(* Logix 5000 project; controller BreakGroup_US vendor 1 type 14 code 211 rev 32.16; software revision 32.05; part 2 of 8 *)

VAR_GLOBAL   (* controller tags *)
   Emg_Stop : BOOL;
   Gantry_01Vertical_Limit_Switch_1 : ALIAS FOR MCP_PT01:23:I.0;
   Gantry_01Vertical_Limit_Switch_2 : ALIAS FOR MCP_PT01:23:I.1;
   Gantry_02_Vertical_Limit_Switch_1 : ALIAS FOR RCP_PT01:22:I.7;
   Gantry_02_Vertical_Limit_Switch_2 : ALIAS FOR RCP_PT01:23:I.0;
   Gantry_1_Clamping_Start_PB : ALIAS FOR MCP_PT01:24:I.5;
   Gantry_1_Clamping_Stop_PB : ALIAS FOR MCP_PT01:24:I.6;
   Gantry_1_EMG_PB : ALIAS FOR MCP_PT01:24:I.0;
   Gantry_1_Gripper_Start : BOOL;
   Gantry_1_Home_PB : ALIAS FOR MCP_PT01:24:I.7;
   Gantry_1_Horizontal_Limit_Switch_01 : ALIAS FOR MCP_PT01:22:I.4;
   Gantry_1_Horizontal_Limit_Switch_02 : ALIAS FOR MCP_PT01:22:I.5;
   Gantry_1_Horizontal_Start : BOOL;
   Gantry_1_Horizontal_Start_PB : ALIAS FOR MCP_PT01:24:I.1;
   Gantry_1_Horizontal_Stop_PB : ALIAS FOR MCP_PT01:24:I.2;
   Gantry_1_LH_Clamping_Limit_Switch_1 : ALIAS FOR MCP_PT01:23:I.2;
   Gantry_1_LH_Clamping_Limit_Switch_2 : ALIAS FOR MCP_PT01:23:I.3;
   Gantry_1_RH_Clamping_Limit_Switch_1 : ALIAS FOR MCP_PT01:23:I.4;
   Gantry_1_RH_Clamping_Limit_Switch_2 : ALIAS FOR MCP_PT01:23:I.5;
   Gantry_1_Vertical_Locking_Cyl_1Extended : ALIAS FOR MCP_PT01:23:I.6;
   Gantry_1_Vertical_Locking_Cyl_1Retracted : ALIAS FOR MCP_PT01:23:I.7;
   Gantry_1_Vertical_Start : BOOL;
   Gantry_1_Vertical_Start_PB : ALIAS FOR MCP_PT01:24:I.3;
   Gantry_1_Vertical_Stop_PB : ALIAS FOR MCP_PT01:24:I.4;
   Gantry_1Collision_sensor : ALIAS FOR MCP_PT01:22:I.6;
   Gantry_1Zero_Pos_Sensor : ALIAS FOR MCP_PT01:22:I.7;
   Gantry_2_Clamping_Start_PB : ALIAS FOR RCP_PT01:24:I.6;
   Gantry_2_Clamping_Stop_PB : ALIAS FOR RCP_PT01:24:I.7;
   Gantry_2_Collision_sensor : ALIAS FOR RCP_PT01:22:I.5;
   Gantry_2_Emg_PB : ALIAS FOR RCP_PT01:24:I.1;
   Gantry_2_Gripper_Start : BOOL;
   Gantry_2_Horizontal_Limit_Switch_01 : ALIAS FOR RCP_PT01:22:I.3;
   Gantry_2_Horizontal_Limit_Switch_02 : ALIAS FOR RCP_PT01:22:I.4;
   Gantry_2_Horizontal_Start : BOOL;
   Gantry_2_Horizontal_Start_PB : ALIAS FOR RCP_PT01:24:I.2;
   Gantry_2_Horizontal_Stop_PB : ALIAS FOR RCP_PT01:24:I.3;
   Gantry_2_LH_Clamping_Limit_Switch_1 : ALIAS FOR RCP_PT01:23:I.1;
   Gantry_2_LH_Clamping_Limit_Switch_2 : ALIAS FOR RCP_PT01:23:I.2;
   Gantry_2_LH_Tilting_Home_PositionSensor : ALIAS FOR RCP_PT01:23:I.7;
   Gantry_2_RH_Clamping_Limit_Switch_1 : ALIAS FOR RCP_PT01:23:I.3;
   Gantry_2_RH_Clamping_Limit_Switch_2 : ALIAS FOR RCP_PT01:23:I.4;
   Gantry_2_RH_Tilting_Home_PositionSensor : ALIAS FOR RCP_PT01:24:I.0;
   Gantry_2_Tilter_LH_Start : BOOL;
   Gantry_2_Tilter_RH_Start : BOOL;
   Gantry_2_Vertical_Locking_Cyl_1Extended : ALIAS FOR RCP_PT01:23:I.5;
   Gantry_2_Vertical_Locking_Cyl_1Retracted : ALIAS FOR RCP_PT01:23:I.6;
   Gantry_2_vertical_Start : BOOL;
   Gantry_2_Vertical_Start_PB : ALIAS FOR RCP_PT01:24:I.4;
   Gantry_2_Vertical_Stop_PB : ALIAS FOR RCP_PT01:24:I.5;
   Gantry_2_Zero_Pos_Sensor : ALIAS FOR RCP_PT01:22:I.6;
   HMI_ACK : BOOL;
   HMI_Gantry_01_Gripper_PB : SINT;
   HMI_Gantry_01_Hor_PB : SINT;
   HMI_Gantry_01_Ver_PB : SINT;
   HMI_Gantry_02_Hor_PB : SINT;
        .0   // Gantry_02_horizontal axis servo enable
        .1   // gantry 2 horizontal axis jog mode selected
        .2   // gantry 2 horizontal axis abs mode selected
        .3   // gantry 2 horizontal axis rel mode selected
        .4   // gantry 2 horizontal start command
        .5   // gantry 2 horizontal axis jog forward cmnd
        .6   // gantry 2 horizontal axis jog reverse cmnd
   HMI_Gantry_2_gripper_PB : SINT;
        .0   // Gantry_2_gripper axis servo enable
        .1   // Gantry_2_gripper axis jog mode selected
        .2   // Gantry_2_gripper axis pos mode selected
        .3   // Gantry_2_gripper axis rel mode selected
        .4   // Gantry_2_gripper axis start command
        .5   // Gantry_2_gripper axis jog forward command
        .6   // Gantry_2_gripper axis jog reverse command
   HMI_Gantry_2_Tilter_LH_PB : SINT;
        .0   // Gantry_2_Tilter_LH axis servo enable
        .1   // Gantry_2_Tilter_LH axis jog mode selected
        .2   // Gantry_2_Tilter_LH axis pos mode selected
        .3   // Gantry_2_Tilter_LH axis rel mode selected
        .4   // Gantry_2_Tilter_LH axis start command
        .5   // Gantry_2_Tilter_LH axis jog forward command
        .6   // Gantry_2_Tilter_LH axis jog reverse command
   HMI_Gantry_2_Tilter_RH_PB : SINT;
        .0   // Gantry_2_Tilter_RH axis servo enable
        .1   // Gantry_2_Tilter_RH axis jog mode selected
        .2   // Gantry_2_Tilter_RH pos mode selected
        .3   // Gantry_2_Tilter_RH rel mode selected
        .4   // Gantry_2_Tilter_RH axis start command
        .5   // Gantry_2_Tilter_RH axis jog forward command
        .6   // Gantry_2_Tilter_RH axis jog rev command
   HMI_Gantry_2_vertical_PB : SINT;
        .0   // Gantry_2_vertical axis servo enable
        .1   // Gantry_2_vertical axis jog mode selected
        .2   // Gantry_2_vertical axis pos mode selected
        .3   // Gantry_2_vertical axis rel mode selected
        .4   // Gantry_2_vertical start command
        .5   // Gantry_2_vertical axis jog forward command
        .6   // Gantry_2_vertical axis jog reverse command
   HMI_MAN_GTY1_GRI_STOP : BOOL;
   HMI_MAN_GTY1_HORIZ_STOP : BOOL;
   HMI_MAN_GTY1_VERT_STOP : BOOL;
   HMI_MAN_GTY2_GRI_STOP : BOOL;
   HMI_MAN_GTY2_HORI_STOP : BOOL;
   HMI_MAN_GTY2_TIL1_STOP : BOOL;
   HMI_MAN_GTY2_TIL2_STOP : BOOL;
   HMI_MAN_GTY2_VERT_STOP : BOOL;
   HMI_MAN_LH_OIL_STOP : BOOL;
   HMI_MAN_RH_OIL_STOP : BOOL;
   HMI_MAN_STN_100_STOP : BOOL;
   HMI_MAN_STN_110_STOP : BOOL;
   HMI_MAN_STN_120_STOP : BOOL;
   HMI_MAN_STN_30_STOP : BOOL;
   HMI_MAN_STN_40_STOP : BOOL;
   HMI_MAN_STN_50_STOP : BOOL;
   HMI_MAN_STN_60_STOP : BOOL;
   HMI_MAN_STN_70_STOP : BOOL;
   HMI_MAN_STN_80_STOP : BOOL;
   HMI_MAN_STN_90_STOP : BOOL;
   HMI_Oil_Tank_LH_PB : SINT;
   HMI_Oil_Tank_RH_PB : SINT;
   HMI_STN30_GRI_SETPOINT : REAL := 300.0;
   HMI_STN30_HORIZ_MOVE_SETPOINT : REAL := 2000.0;
   HMI_STN30_VER_LIFTUP_SETPOINT : REAL := 10.0;
   HMI_STN30_VER_PICK_SETPOINT : REAL := 50.0;
   HMI_STN40_GRI_GRIP_POINT : REAL;
   HMI_STN40_GRI_SETPOINT : REAL := 200.0;
   HMI_STN40_HORIZ_MOVE_SETPOINT : REAL := 1000.0;
   HMI_STN40_VER_LIFTUP_SETPOINT : REAL := 10.0;
   HMI_STN40_VER_PICK_LIFTUP_SETPOINT : REAL;
   HMI_STN40_VER_PICK_SETPOINT : REAL := 50.0;
   HMI_STN40_VER_PLACE_SETPOINT : REAL;
   HMI_STN50_DE_GRIPPER_SETPOINT : REAL;
   HMI_STN50_GRI_GRIP_POINT : REAL;
   HMI_STN50_HORIZ_MOVE_SETPOINT : REAL;
   HMI_STN50_VER_DROP_SETPOINT : REAL;
   HMI_STN50_VER_LIFTUP_SETPOINT : REAL;
   HMI_STN50_VER_PICK_LIFTUP_SETPOINT : REAL;
   HMI_STN50_VER_PICK_SETPOINT : DINT;
   MAN_GTY1_GRI_HOME : TIMER := (PRE := 1000);
   MAN_GTY1_HORI_HOME : TIMER := (PRE := 1000);
   MAN_GTY1_VERT_HOME : TIMER := (PRE := 1000);
   MAN_GTY2_GRI_HOME : TIMER := (PRE := 1000);
   MAN_GTY2_HORI_HOME : TIMER := (PRE := 1000);
   MAN_GTY2_TIL1_HOME : TIMER := (PRE := 1000);
   MAN_GTY2_TIL2_HOME : TIMER := (PRE := 1000);
   MAN_GTY2_VERT_HOME : TIMER := (PRE := 1000);
   MAN_LH_OIL_TIME : TIMER := (PRE := 1000);
   MAN_RH_OIL_TIME : TIMER := (PRE := 1000);
   MAN_STN_100_HOME : TIMER := (PRE := 1000);
   MAN_STN_110_HOME : TIMER := (PRE := 1000);
   MAN_STN_120_HOME : TIMER := (PRE := 1000);
   MAN_STN_30_HOME : TIMER := (PRE := 1000);
   MAN_STN_40_HOME : TIMER := (PRE := 1000);
   MAN_STN_50_HOME : TIMER := (PRE := 1000);
   man_STN_60_HOME : TIMER := (PRE := 1000);
   MAN_STN_70_HOME : TIMER := (PRE := 1000);
   MAN_STN_80_HOME : TIMER := (PRE := 1000);
   MAN_STN_90_HOME : TIMER := (PRE := 1000);
   MCP_GY_01_Gripper : MCP_Servo_01 := (Inverter_Ready := 1, STO_InActive := 1, Referenced_Drive := 1, Status_Suberror_Num := 13, Digital_Inputs := 2#0000_0000_0000_0001, Actual_Mode := 400, Actual_Pos := 331.5, Enable_EsTop := 1, Speed := 10.0, Accel_Ramp := 30.0, Decel_Ramp := 30.0, Application_Mode := 400, Target_Position := 331.5, PositionDecimal_Place := 2);
   MCP_GY_01_Horizontal : MCP_Servo_02 := (Start_Offest_Num := 16, Inverter_Ready := 1, STO_InActive := 1, Referenced_Drive := 1, SftWreLiMits_DisAble := 1, Status_Suberror_Num := 13, Digital_Inputs := 2#0000_0000_0000_0001, Actual_Mode := 400, Actual_Pos := 6159.3, Enable_EsTop := 1, Speed := 20.0, Accel_Ramp := 100.0, Decel_Ramp := 100.0, Application_Mode := 400, Target_Position := 6159.3, PositionDecimal_Place := 2);
   MCP_GY_01_Vertical : MCP_Servo_02 := (Start_Offest_Num := 8, Inverter_Ready := 1, STO_InActive := 1, Referenced_Drive := 1, Status_Suberror_Num := 13, Digital_Inputs := 2#0000_0000_0000_0001, Actual_Mode := 400, Actual_Pos := 570.8, Enable_EsTop := 1, Speed := 10.0, Accel_Ramp := 50.0, Decel_Ramp := 50.0, Application_Mode := 400, Target_Position := 570.8, PositionDecimal_Place := 2);
   MCP_IO : DINT[7];
   MCP_ST_30_Turntable_Motor : MCP_Servo_02 := (Start_Offest_Num := 64, Inverter_Ready := 1, STO_InActive := 1, Referenced_Drive := 1, SftWreLiMits_DisAble := 1, Status_Suberror_Num := 13, Digital_Inputs := 2#0000_0000_0000_0001, Actual_Mode := 400, Enable_EsTop := 1, Speed := 10.0, Accel_Ramp := 30.0, Decel_Ramp := 30.0, Application_Mode := 400, PositionDecimal_Place := 2);
   MCP_ST_40_Turntable_Motor : MCP_Servo_02 := (Start_Offest_Num := 56, Inverter_Ready := 1, STO_InActive := 1, Referenced_Drive := 1, SftWreLiMits_DisAble := 1, Status_Suberror_Num := 13, Digital_Inputs := 2#0000_0000_0000_0001, Actual_Mode := 100, Enable_EsTop := 1, Application_Mode := 100, PositionDecimal_Place := 2);
   MCP_ST_50_Turntable_Motor : MCP_Servo_02 := (Start_Offest_Num := 48, Inverter_Ready := 1, STO_InActive := 1, Referenced_Drive := 1, SftWreLiMits_DisAble := 1, Status_Suberror_Num := 13, Digital_Inputs := 2#0000_0000_0000_0001, Actual_Mode := 400, Enable_EsTop := 1, Speed := 10.0, Accel_Ramp := 30.0, Decel_Ramp := 30.0, Application_Mode := 400, Target_Position := 180.0, PositionDecimal_Place := 2);
   MCP_ST_60_Turntable_Motor : MCP_Servo_02 := (Start_Offest_Num := 40, Inverter_Ready := 1, STO_InActive := 1, SftWreLiMits_DisAble := 1, Status_Suberror_Num := 13, Digital_Inputs := 2#0000_0000_0000_0001, Actual_Mode := 100, Actual_Pos := 524.44, Enable_EsTop := 1, Application_Mode := 100, PositionDecimal_Place := 2);
   MCP_ST_70_Turntable_Motor : MCP_Servo_02 := (Start_Offest_Num := 32, STO_InActive := 1, SftWreLiMits_DisAble := 1, Status_Suberror_Num := 1, Digital_Inputs := 2#0000_0000_0000_0001, Actual_Mode := 100, Enable_EsTop := 1, Application_Mode := 100, PositionDecimal_Place := 2);
   MCP_ST_80_Turntable_Motor : MCP_Servo_02 := (Start_Offest_Num := 24, Inverter_Ready := 1, STO_InActive := 1, Referenced_Drive := 1, SftWreLiMits_DisAble := 1, Status_Suberror_Num := 13, Digital_Inputs := 2#0000_0000_0000_0001, Actual_Mode := 100, Actual_Pos := 80.42, Enable_EsTop := 1, Speed := 10.0, Accel_Ramp := 30.0, Decel_Ramp := 30.0, Application_Mode := 100, PositionDecimal_Place := 2);
   Out_ST30_Home_PB : ALIAS FOR MCP_PT01:26:O.7;
   Out_ST30_Hydro_Motor_On : ALIAS FOR MCP_PT01:26:O.4;
   Out_ST30_Index_PlateLockCyl1_Extend : ALIAS FOR MCP_PT01:25:O.4;
   Out_ST30_Index_PlateLockCyl1_Retract : ALIAS FOR MCP_PT01:25:O.5;
   Out_ST30_Index_PlateLockCyl2_Extend : ALIAS FOR MCP_PT01:25:O.6;
   Out_ST30_Index_PlateLockCyl2_Retract : ALIAS FOR MCP_PT01:25:O.7;
   Out_ST30_Press_Unit_Cyl_1Extend : ALIAS FOR MCP_PT01:26:O.0;
   Out_ST30_Press_Unit_Cyl_1Retract : ALIAS FOR MCP_PT01:26:O.1;
   Out_ST30_Press_Unit_Cyl_2Extend : ALIAS FOR MCP_PT01:26:O.2;
   Out_ST30_Press_Unit_Cyl_2Retract : ALIAS FOR MCP_PT01:26:O.3;
   Out_ST30_Reset_PB : ALIAS FOR MCP_PT01:27:O.0;
   Out_ST30_Servo_Healthy_Indication : ALIAS FOR MCP_PT01:27:O.1;
   Out_ST30_Servo_Trip_Indication : ALIAS FOR MCP_PT01:27:O.2;
   Out_ST30_Start_PB : ALIAS FOR MCP_PT01:26:O.5;
   Out_ST30_Stop_PB : ALIAS FOR MCP_PT01:26:O.6;
   Out_ST40_Home_PB : ALIAS FOR MCP_PT01:30:O.6;
   Out_ST40_Index_PlateLockCyl1_Extend : ALIAS FOR MCP_PT01:27:O.3;
   Out_ST40_Index_PlateLockCyl1_Retract : ALIAS FOR MCP_PT01:27:O.4;
   Out_ST40_Index_PlateLockCyl2_Extend : ALIAS FOR MCP_PT01:27:O.5;
   Out_ST40_Index_PlateLockCyl2_Retract : ALIAS FOR MCP_PT01:27:O.6;
   Out_ST40_Reset_PB : ALIAS FOR MCP_PT01:30:O.7;
   Out_ST40_Servo_Healthy_Indication : ALIAS FOR MCP_PT01:31:O.0;
   Out_ST40_Servo_Trip_Indication : ALIAS FOR MCP_PT01:31:O.1;
   Out_ST40_Start_PB : ALIAS FOR MCP_PT01:30:O.4;
   Out_ST40_Stop_PB : ALIAS FOR MCP_PT01:30:O.5;
   Out_ST_10_Trolley_1LockCylExtend : ALIAS FOR MCP_PT01:25:O.0;
   Out_ST_10_Trolley_1LockCylRetract : ALIAS FOR MCP_PT01:25:O.1;
   Out_ST_20_Trolley_1LockCylExtend : ALIAS FOR MCP_PT01:25:O.2;
   Out_ST_20_Trolley_1LockCylRetract : ALIAS FOR MCP_PT01:25:O.3;
   RCP_GY_02_Gripper : RCP_Servo_01 := (Inverter_Ready := 1, STO_InActive := 1, Referenced_Drive := 1, SftWreLiMits_DisAble := 1, Status_Suberror_Num := 1, Actual_Mode := 100, Actual_Pos := 450.0, Enable_EsTop := 1, Application_Mode := 100, PositionDecimal_Place := 2);
   RCP_GY_02_Horizontal : RCP_Servo_02 := (Start_Offest_Num := 16, Inverter_Ready := 1, STO_InActive := 1, Referenced_Drive := 1, SftWreLiMits_DisAble := 1, Status_Suberror_Num := 13, Digital_Inputs := 2#0000_0000_0000_0001, Actual_Mode := 100, Enable_EsTop := 1, Application_Mode := 100, PositionDecimal_Place := 2);
   RCP_GY_02_Vertical : RCP_Servo_02 := (Start_Offest_Num := 8, Inverter_Ready := 1, STO_InActive := 1, Referenced_Drive := 1, SftWreLiMits_DisAble := 1, Status_Suberror_Num := 1, Actual_Mode := 100, Enable_EsTop := 1, Application_Mode := 100, PositionDecimal_Place := 2);
   RCP_LH_Oil_Tank_Lift : RCP_Servo_02 := (Start_Offest_Num := 24, Inverter_Ready := 1, STO_InActive := 1, SftWreLiMits_DisAble := 1, Status_Suberror_Num := 13, Digital_Inputs := 2#0000_0000_0000_0001, Actual_Mode := 100, Actual_Pos := -11.36, Enable_EsTop := 1, Application_Mode := 100, PositionDecimal_Place := 2);
   RCP_LH_Oil_Tank_Lift_Start : BOOL;
   RCP_RH_Oil_Tank_Lift : RCP_Servo_02 := (Start_Offest_Num := 32, Inverter_Ready := 1, STO_InActive := 1, SftWreLiMits_DisAble := 1, Status_Suberror_Num := 13, Digital_Inputs := 2#0000_0000_0000_0001, Actual_Mode := 100, Actual_Pos := -17.5, Enable_EsTop := 1, Application_Mode := 100, PositionDecimal_Place := 2);
   RCP_RH_Oil_Tank_Lift_Start : BOOL;
   RCP_ST_100_Turntable_Motor : RCP_Servo_02 := (Start_Offest_Num := 88, Inverter_Ready := 1, STO_InActive := 1, Referenced_Drive := 1, SftWreLiMits_DisAble := 1, Status_Suberror_Num := 13, Digital_Inputs := 2#0000_0000_0000_0001, Actual_Mode := 100, Enable_EsTop := 1, Application_Mode := 100, PositionDecimal_Place := 2);
   RCP_ST_110_Turntable_Motor : RCP_Servo_02 := (Start_Offest_Num := 40, Inverter_Ready := 1, STO_InActive := 1, Referenced_Drive := 1, SftWreLiMits_DisAble := 1, Status_Suberror_Num := 13, Digital_Inputs := 2#0000_0000_0000_0001, Actual_Mode := 100, Enable_EsTop := 1, Application_Mode := 100, PositionDecimal_Place := 2);
   RCP_ST_120_Turntable_Motor : RCP_Servo_02 := (Start_Offest_Num := 48, Inverter_Ready := 1, STO_InActive := 1, SftWreLiMits_DisAble := 1, Status_Suberror_Num := 13, Digital_Inputs := 2#0000_0000_0000_0001, Actual_Mode := 100, Actual_Pos := 15.66, Enable_EsTop := 1, Application_Mode := 100, PositionDecimal_Place := 2);
   RCP_ST_60_Conveyor_Motor : RCP_Servo_02 := (Start_Offest_Num := 72, Inverter_Ready := 1, STO_InActive := 1, SftWreLiMits_DisAble := 1, Status_Suberror_Num := 13, Digital_Inputs := 2#0000_0000_0000_0001, Actual_Pos := -15113.0, Enable_EsTop := 1);
   RCP_ST_90_Conveyor_Motor : RCP_Servo_02 := (Start_Offest_Num := 72, STO_InActive := 1, Fault_Active := 1, SftWreLiMits_DisAble := 1, Fault_Num := 26, Status_Suberror_Num := 2, Digital_Inputs := 2#0000_0000_0000_0001, Actual_Mode := 100, Actual_Pos := -16.96, Enable_EsTop := 1, Application_Mode := 100, PositionDecimal_Place := 2);
   RCP_ST_90_Turntable_Motor : RCP_Servo_02 := (Start_Offest_Num := 80, Inverter_Ready := 1, STO_InActive := 1, Referenced_Drive := 1, SftWreLiMits_DisAble := 1, Status_Suberror_Num := 13, Digital_Inputs := 2#0000_0000_0000_0001, Actual_Mode := 300, Enable_EsTop := 1, Speed := 10.0, Accel_Ramp := 10.0, Decel_Ramp := 10.0, Application_Mode := 300, PositionDecimal_Place := 2);
   RCP_Tilt_Axis_Master : RCP_Servo_02 := (Start_Offest_Num := 56, Inverter_Ready := 1, STO_InActive := 1, Referenced_Drive := 1, SftWreLiMits_DisAble := 1, Status_Suberror_Num := 13, Digital_Inputs := 2#0000_0000_0000_0001, Actual_Mode := 100, Actual_Pos := 1800.0, Enable_EsTop := 1, Application_Mode := 100, PositionDecimal_Place := 2);
   RCP_Tilt_Axis_Slave : RCP_Servo_02 := (Start_Offest_Num := 64, Inverter_Ready := 1, STO_InActive := 1, Referenced_Drive := 1, Warning_Active := 1, SftWreLiMits_DisAble := 1, Status_Suberror_Num := 13, Digital_Inputs := 2#0000_0000_0000_0001, Actual_Mode := 100, Actual_Pos := 100.0, Enable_EsTop := 1, Application_Mode := 100, PositionDecimal_Place := 2);
   ST : BOOL;
   ST100_Auto_SS : ALIAS FOR RCP_PT01:14:I.3;
   ST100_Conv_End_Sensor : ALIAS FOR RCP_PT01:10:I.7;
   ST100_Conv_Home_Sensor : ALIAS FOR RCP_PT01:10:I.6;
   ST100_EMG_PB : ALIAS FOR RCP_PT01:13:I.5;
   ST100_Home_PB : ALIAS FOR RCP_PT01:14:I.2;
   ST100_IndexPlateLockCyl01_Extended : ALIAS FOR RCP_PT01:10:I.2;
   ST100_IndexPlateLockCyl01_Retracted : ALIAS FOR RCP_PT01:10:I.3;
   ST100_IndexPlateLockCyl02_Extended : ALIAS FOR RCP_PT01:10:I.4;
   ST100_IndexPlateLockCyl02_Retracted : ALIAS FOR RCP_PT01:10:I.5;
   ST100_IndexTableHomePositionSensor : ALIAS FOR RCP_PT01:10:I.1;
   ST100_Manual_SS : ALIAS FOR RCP_PT01:14:I.4;
   ST100_Product_Present_Sensor : ALIAS FOR RCP_PT01:10:I.0;
   ST100_Reset_PB : ALIAS FOR RCP_PT01:14:I.5;
   ST100_Start_1_PB : ALIAS FOR RCP_PT01:13:I.6;
   ST100_Start_2_PB : ALIAS FOR RCP_PT01:14:I.0;
   ST100_Stop_1_PB : ALIAS FOR RCP_PT01:13:I.7;
   ST100_Stop_2_PB : ALIAS FOR RCP_PT01:14:I.1;
   ST10_Pre_Condition_OK : BOOL;
   ST10_Trolley1Lock_Cyl_01_Extended : ALIAS FOR MCP_PT01:1:I.0;
   ST10_Trolley1LockCyl_01_Retracted : ALIAS FOR MCP_PT01:1:I.1;
   ST10_Trolley_Present_Sensor : ALIAS FOR MCP_PT01:1:I.2;
   ST10_TrolleyTopSideProductPresentSensor : ALIAS FOR MCP_PT01:1:I.3;
   ST110_Auto_SS : ALIAS FOR RCP_PT01:17:I.2;
   ST110_Conv_End_Sensor : ALIAS FOR RCP_PT01:15:I.5;
   ST110_Conv_Home_Sensor : ALIAS FOR RCP_PT01:15:I.4;
   ST110_EMG_PB : ALIAS FOR RCP_PT01:16:I.4;
   ST110_Home_PB : ALIAS FOR RCP_PT01:17:I.1;
   ST110_IndexPlateLockCyl01_Extended : ALIAS FOR RCP_PT01:15:I.0;
   ST110_IndexPlateLockCyl01_Retracted : ALIAS FOR RCP_PT01:15:I.1;
   ST110_IndexPlateLockCyl02_Extended : ALIAS FOR RCP_PT01:15:I.2;
   ST110_IndexPlateLockCyl02_Retracted : ALIAS FOR RCP_PT01:15:I.3;
   ST110_IndexTableHomePositionSensor : ALIAS FOR RCP_PT01:14:I.7;
   ST110_Manual_SS : ALIAS FOR RCP_PT01:17:I.3;
   ST110_Product_Present_Sensor : ALIAS FOR RCP_PT01:14:I.6;
   ST110_Reset_PB : ALIAS FOR RCP_PT01:17:I.4;
   ST110_Start_1_PB : ALIAS FOR RCP_PT01:16:I.5;
   ST110_Start_2_PB : ALIAS FOR RCP_PT01:16:I.7;
   ST110_Stop_1_PB : ALIAS FOR RCP_PT01:16:I.6;
   ST110_Stop_2_PB : ALIAS FOR RCP_PT01:17:I.0;
   ST120_Auto_SS : ALIAS FOR RCP_PT01:22:I.0;
   ST120_Conv_End_Sensor : ALIAS FOR RCP_PT01:18:I.4;
   ST120_Conv_Home_Sensor : ALIAS FOR RCP_PT01:18:I.3;
   ST120_EMG_PB : ALIAS FOR RCP_PT01:21:I.2;
   ST120_Home_PB : ALIAS FOR RCP_PT01:21:I.7;
   ST120_IndexPlateLockCyl01_Extended : ALIAS FOR RCP_PT01:17:I.7;
   ST120_IndexPlateLockCyl01_Retracted : ALIAS FOR RCP_PT01:18:I.0;
   ST120_IndexPlateLockCyl02_Extended : ALIAS FOR RCP_PT01:18:I.1;
   ST120_IndexPlateLockCyl02_Retracted : ALIAS FOR RCP_PT01:18:I.2;
   ST120_IndexTableHomePositionSensor : ALIAS FOR RCP_PT01:17:I.6;
   ST120_Manual_SS : ALIAS FOR RCP_PT01:22:I.1;
   ST120_Product_Present_Sensor : ALIAS FOR RCP_PT01:17:I.5;
   ST120_Reset_PB : ALIAS FOR RCP_PT01:22:I.2;
   ST120_Start_1_PB : ALIAS FOR RCP_PT01:21:I.3;
   ST120_Start_2_PB : ALIAS FOR RCP_PT01:21:I.5;
   ST120_Stop_1_PB : ALIAS FOR RCP_PT01:21:I.4;
   ST120_Stop_2_PB : ALIAS FOR RCP_PT01:21:I.6;
   ST20_Trolley_Present_Sensor_02 : ALIAS FOR MCP_PT01:1:I.6;
   ST20_TrolleyTopSideProductPresentSensor : ALIAS FOR MCP_PT01:4:I.3;
   ST30_Auto_SS : ALIAS FOR MCP_PT01:6:I.3;
   ST30_Emg_Push_Buttion : ALIAS FOR MCP_PT01:5:I.7;
   ST30_Home_PB : ALIAS FOR MCP_PT01:6:I.2;
   ST30_Hydro_motor : ALIAS FOR MCP_PT01:5:I.6;
   ST30_IndexingTableHomePositionSensor : ALIAS FOR MCP_PT01:4:I.5;
   ST30_IndexPlateLockCyl1Extended : ALIAS FOR MCP_PT01:4:I.6;
   ST30_IndexPlateLockCyl1Retracted : ALIAS FOR MCP_PT01:4:I.7;
   ST30_IndexPlateLockCyl2Extended : ALIAS FOR MCP_PT01:5:I.0;
   ST30_IndexPlateLockCyl2Retracted : ALIAS FOR MCP_PT01:5:I.1;
   ST30_MAN_PB : SINT;
        .0   // ST30_Servo_Enable
        .1   // ST30_Jog_Mode
        .2   // ST30_POS_Mode
        .3   // ST30_REL_Mode
        .4   // ST30_Start
        .5   // ST30_Jog_FWD
        .6   // ST30_Jog_REV
   ST30_Manual_SS : ALIAS FOR MCP_PT01:6:I.4;
   ST30_PressUnitCyl_1Extended : ALIAS FOR MCP_PT01:5:I.2;
   ST30_PressUnitCyl_1Retracted : ALIAS FOR MCP_PT01:5:I.3;
   ST30_PressUnitCyl_2Extended : ALIAS FOR MCP_PT01:5:I.4;
   ST30_PressUnitCyl_2Retracted : ALIAS FOR MCP_PT01:5:I.5;
   ST30_Product_Present_Sensor : ALIAS FOR MCP_PT01:4:I.4;
   ST30_Reset_PB : ALIAS FOR MCP_PT01:6:I.5;
   ST30_Start : BOOL;
   ST30_Start_PB : ALIAS FOR MCP_PT01:6:I.0;
   ST30_Stop_PB : ALIAS FOR MCP_PT01:6:I.1;
   ST40_Auto_SS : ALIAS FOR MCP_PT01:10:I.5;
   ST40_EMG_PB : ALIAS FOR MCP_PT01:10:I.1;
   ST40_Home_PB : ALIAS FOR MCP_PT01:10:I.4;
   ST40_IndexingTableHomePositionSensor : ALIAS FOR MCP_PT01:6:I.7;
   ST40_IndexPlateLockCyl01_Extended : ALIAS FOR MCP_PT01:7:I.0;
   ST40_IndexPlateLockCyl01_Retracted : ALIAS FOR MCP_PT01:7:I.1;
   ST40_IndexPlateLockCyl02_Extended : ALIAS FOR MCP_PT01:7:I.2;
   ST40_IndexPlateLockCyl02_Retracted : ALIAS FOR MCP_PT01:7:I.3;
   ST40_Manual_SS : ALIAS FOR MCP_PT01:10:I.6;
   ST40_ProductPresentSensor : ALIAS FOR MCP_PT01:6:I.6;
   ST40_Reset_PB : ALIAS FOR MCP_PT01:10:I.7;
   ST40_Start_PB : ALIAS FOR MCP_PT01:10:I.2;
   ST40_Stop_PB : ALIAS FOR MCP_PT01:10:I.3;
   ST50_Auto_SS : ALIAS FOR MCP_PT01:15:I.1;
   ST50_Conv_End_Sensor : ALIAS FOR MCP_PT01:11:I.7;
   ST50_Conv_Home_Sensor : ALIAS FOR MCP_PT01:11:I.6;
   ST50_EMG_PB : ALIAS FOR MCP_PT01:14:I.5;
   ST50_Home_PB : ALIAS FOR MCP_PT01:15:I.0;
   ST50_IndexPlateLockCyl01_Extended : ALIAS FOR MCP_PT01:11:I.2;
   ST50_IndexPlateLockCyl01_Retracted : ALIAS FOR MCP_PT01:11:I.3;
   ST50_IndexPlateLockCyl02_Extended : ALIAS FOR MCP_PT01:11:I.4;
   ST50_IndexPlateLockCyl02_Retracted : ALIAS FOR MCP_PT01:11:I.5;
   ST50_IndexTableHomePositionSensor : ALIAS FOR MCP_PT01:11:I.1;
   ST50_Manual_SS : ALIAS FOR MCP_PT01:15:I.2;
   ST50_Product_Present_Sensor : ALIAS FOR MCP_PT01:11:I.0;
   ST50_Reset_PB : ALIAS FOR MCP_PT01:15:I.3;
   ST50_Start_PB : ALIAS FOR MCP_PT01:14:I.6;
   ST50_Stop_PB : ALIAS FOR MCP_PT01:14:I.7;
   ST60_Auto_SS : ALIAS FOR MCP_PT01:20:I.2;
   ST60_Conv_End_Sensor : ALIAS FOR MCP_PT01:16:I.3;
   ST60_Conv_Home_Sensor : ALIAS FOR MCP_PT01:16:I.2;
   ST60_EMG_PB : ALIAS FOR MCP_PT01:19:I.6;
   ST60_Home_PB : ALIAS FOR MCP_PT01:20:I.1;
   ST60_Hydro_Motor : ALIAS FOR MCP_PT01:17:I.0;
   ST60_IndexPlateLockCyl01_Extended : ALIAS FOR MCP_PT01:15:I.6;
   ST60_IndexPlateLockCyl01_Retracted : ALIAS FOR MCP_PT01:15:I.7;
   ST60_IndexPlateLockCyl02_Extended : ALIAS FOR MCP_PT01:16:I.0;
   ST60_IndexPlateLockCyl02_Retracted : ALIAS FOR MCP_PT01:16:I.1;
   ST60_IndexTableHomePositionSensor : ALIAS FOR MCP_PT01:15:I.5;
   ST60_Manual_SS : ALIAS FOR MCP_PT01:20:I.3;
   ST60_Press_Unit_Cyl01_Extended : ALIAS FOR MCP_PT01:16:I.4;
   ST60_Press_Unit_Cyl01_Retracted : ALIAS FOR MCP_PT01:16:I.5;
   ST60_Press_Unit_Cyl02_Extended : ALIAS FOR MCP_PT01:16:I.6;
   ST60_Press_Unit_Cyl02_Retracted : ALIAS FOR MCP_PT01:16:I.7;
   ST60_Product_Present_Sensor : ALIAS FOR MCP_PT01:15:I.4;
   ST60_Reset_PB : ALIAS FOR MCP_PT01:20:I.4;
   ST60_Start_PB : ALIAS FOR MCP_PT01:19:I.7;
   ST60_Stop_PB : ALIAS FOR MCP_PT01:20:I.0;
   ST70_Auto_SS : ALIAS FOR MCP_PT01:22:I.1;
   ST70_Conv_End_Sensor : ALIAS FOR MCP_PT01:21:I.4;
   ST70_Conv_Home_Sensor : ALIAS FOR MCP_PT01:21:I.3;
   ST70_EMG_PB : ALIAS FOR MCP_PT01:21:I.5;
   ST70_Home_PB : ALIAS FOR MCP_PT01:22:I.0;
   ST70_IndexPlateLockCyl01_Extended : ALIAS FOR MCP_PT01:20:I.7;
   ST70_IndexPlateLockCyl01_Retracted : ALIAS FOR MCP_PT01:21:I.0;
   ST70_IndexPlateLockCyl02_Extended : ALIAS FOR MCP_PT01:21:I.1;
   ST70_IndexPlateLockCyl02_Retracted : ALIAS FOR MCP_PT01:21:I.2;
   ST70_IndexTableHomePositionSensor : ALIAS FOR MCP_PT01:20:I.6;
   ST70_Manual_SS : ALIAS FOR MCP_PT01:22:I.2;
   ST70_Product_Present_Sensor : ALIAS FOR MCP_PT01:20:I.5;
   ST70_Reset_PB : ALIAS FOR MCP_PT01:22:I.3;
   ST70_Start_PB : ALIAS FOR MCP_PT01:21:I.6;
   ST70_Stop_PB : ALIAS FOR MCP_PT01:21:I.7;
   ST80_Auto_SS : ALIAS FOR RCP_PT01:6:I.0;
   ST80_Conv_End_Sensor : ALIAS FOR RCP_PT01:1:I.7;
   ST80_Conv_Home_Sensor : ALIAS FOR RCP_PT01:1:I.6;
   ST80_EMG_PB : ALIAS FOR RCP_PT01:5:I.2;
   ST80_Home_PB : ALIAS FOR RCP_PT01:5:I.7;
   ST80_Hydro_Motor : ALIAS FOR RCP_PT01:2:I.4;
   ST80_IndexPlateLockCyl01_Extended : ALIAS FOR RCP_PT01:1:I.2;
   ST80_IndexPlateLockCyl01_Retracted : ALIAS FOR RCP_PT01:1:I.3;
   ST80_IndexPlateLockCyl02_Extended : ALIAS FOR RCP_PT01:1:I.4;
   ST80_IndexPlateLockCyl02_Retracted : ALIAS FOR RCP_PT01:1:I.5;
   ST80_IndexTableHomePositionSensor : ALIAS FOR RCP_PT01:1:I.1;
   ST80_Manual_SS : ALIAS FOR RCP_PT01:6:I.1;
   ST80_Press_Unit_Cyl01_Extended : ALIAS FOR RCP_PT01:2:I.0;
   ST80_Press_Unit_Cyl01_Retracted : ALIAS FOR RCP_PT01:2:I.1;
   ST80_Press_Unit_Cyl02_Extended : ALIAS FOR RCP_PT01:2:I.2;
   ST80_Press_Unit_Cyl02_Retracted : ALIAS FOR RCP_PT01:2:I.3;
   ST80_Product_Present_Sensor : ALIAS FOR RCP_PT01:1:I.0;
   ST80_Reset_PB : ALIAS FOR RCP_PT01:6:I.2;
   ST80_Start_2_PB : ALIAS FOR RCP_PT01:5:I.5;
   ST80_Stop_2_PB : ALIAS FOR RCP_PT01:5:I.6;
   ST90_Auto_SS : ALIAS FOR RCP_PT01:9:I.5;
   ST90_Conv_End_Sensor : ALIAS FOR RCP_PT01:7:I.2;
   ST90_Conv_Home_Sensor : ALIAS FOR RCP_PT01:7:I.1;
   ST90_EMG_PB : ALIAS FOR RCP_PT01:8:I.7;
   ST90_Home_PB : ALIAS FOR RCP_PT01:9:I.4;
   ST90_IndexPlateLockCyl01_Extended : ALIAS FOR RCP_PT01:6:I.5;
   ST90_IndexPlateLockCyl01_Retracted : ALIAS FOR RCP_PT01:6:I.6;
   ST90_IndexPlateLockCyl02_Extended : ALIAS FOR RCP_PT01:6:I.7;
   ST90_IndexPlateLockCyl02_Retracted : ALIAS FOR RCP_PT01:7:I.0;
   ST90_IndexTableHomePositionSensor : ALIAS FOR RCP_PT01:6:I.4;
   ST90_Manual_SS : ALIAS FOR RCP_PT01:9:I.6;
   ST90_Product_Present_Sensor : ALIAS FOR RCP_PT01:6:I.3;
   ST90_Reset_PB : ALIAS FOR RCP_PT01:9:I.7;
   ST90_Start_1_PB : ALIAS FOR RCP_PT01:9:I.0;
   ST90_Start_2_PB : ALIAS FOR RCP_PT01:9:I.2;
   ST90_Stop_1_PB : ALIAS FOR RCP_PT01:9:I.1;
   ST90_Stop_2_PB : ALIAS FOR RCP_PT01:9:I.3;
   ST_100_Start : BOOL;
   ST_10_SEQ : DINT;
   ST_10_T1 : TIMER := (PRE := 1000);
   ST_10_Trolley_FRWD : BOOL;
   ST_110_Start : BOOL;
   ST_120_Start : BOOL;
   ST_20Trolley_1LockCylExtended : ALIAS FOR MCP_PT01:1:I.4;
   ST_20Trolley_1LockingCylRetracted : ALIAS FOR MCP_PT01:1:I.5;
   ST_30_Start : BOOL;
   ST_40_Start : BOOL;
   ST_50_Start : BOOL;
   ST_60_Start : BOOL;
   ST_70_Start : BOOL;
   ST_80_Start : BOOL;
   ST_90_Start : BOOL;
   STN50_T1_01 : TIMER := (PRE := 100);
   STN50_T2_01 : TIMER := (PRE := 100);
   STN50_T3_01 : TIMER := (PRE := 100);
   STN50_T4_01 : TIMER := (PRE := 100);
   STN50_T5_01 : TIMER := (PRE := 100);
   STN50_T6_01 : TIMER := (PRE := 100);
   STN50_T7_01 : TIMER := (PRE := 100);
   STN_100_Connection_Fault : BOOL;
   STN_100_Conveyor : INDEX_Block;
   STN_100_HMI_PB : SINT[2];
   STN_100_INDEXING_Connection : BOOL;
   STN_110_Connection_fault : BOOL;
   STN_110_Conveyor : INDEX_Block;
   STN_110_HMI_PB : SINT[2];
   STN_110_RUN : BOOL;
   STN_120_Connection_fault : BOOL;
   STN_120_Conveyor : INDEX_Block;
   STN_120_HMI_PB : SINT[2];
   STN_30_Auto_ENable : BOOL := 1;
   STN_30_HMI_PB : SINT;
   STN_30_PRE_COND_OK : BOOL;
   STN_30_SEQ : DINT := 10;
   STN_30_SEQUENCE_AUTO : SINT;
        .0   // Vertical pick point start
        .1   // Gripper close start
        .2   // vertical home point start
        .3   // horizontal next stn point start
   STN_40_HMI_PB : SINT;
   STN_40_PRE_COND_OK : BOOL;
   STN_40_SEQ : DINT;
   STN_40_SEQUENCE_AUTO : SINT;
        .0   // vertical drop point start
        .1   // gripper release point start
        .2   // vertical home point start
        .3   // horizontal next point start
   STN_50_Conveyor : INDEX_Block := (COMMUNICATION_OK := 1);
   STN_50_Conveyor_Connection_Fault : BOOL;
   STN_50_HMI_PB : SINT[2] := ([0] := 2);
   STN_50_SEQ : DINT;
   STN_50_SEQUENCE_AUTO : SINT;
   STN_60_Conveyor : INDEX_Block;
   STN_60_HMI_PB : SINT[2];
   STN_70_HMI_PB : SINT[2];
   STN_80_HMI_PB : SINT[2];
   STN_90_HMI_PB : SINT[2];
   T10_01 : TIMER := (PRE := 100);
   T11_01 : TIMER := (PRE := 100);
   T1_01 : TIMER := (PRE := 100);
   T2_01 : TIMER := (PRE := 100);
   T3_01 : TIMER := (PRE := 100);
   T4_01 : TIMER := (PRE := 100);
   T5_01 : TIMER := (PRE := 100);
   T6_01 : TIMER := (PRE := 100);
   T7_01 : TIMER := (PRE := 100);
   T8_01 : TIMER := (PRE := 100);
   T9_01 : TIMER := (PRE := 100);
   tEST_012 : BOOL;
   TEST_02 : BOOL;
   Test_COND_OK : DINT;
END_VAR

PROGRAM Gantry_01_Gripper   (* main routine Main *)

ROUTINE Main   (* ladder *)
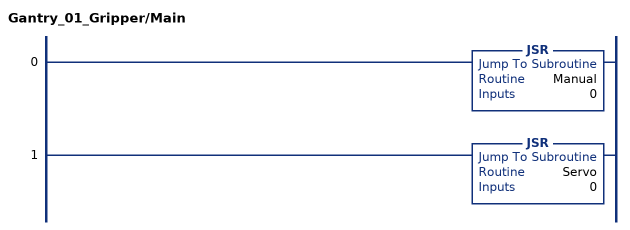
   0: JSR(Manual,0);
   1: JSR(Servo,0);
END_ROUTINE

ROUTINE Manual   (* ladder *)
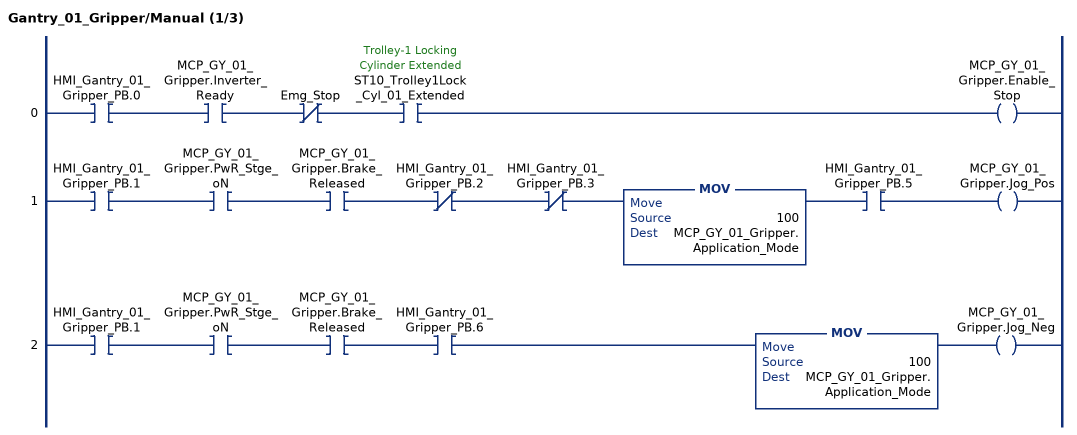
   0: XIC(HMI_Gantry_01_Gripper_PB.0)XIC(MCP_GY_01_Gripper.Inverter_Ready)XIO(Emg_Stop)XIC(ST10_Trolley1Lock_Cyl_01_Extended)OTE(MCP_GY_01_Gripper.Enable_Stop);
   1: XIC(HMI_Gantry_01_Gripper_PB.1)XIC(MCP_GY_01_Gripper.PwR_Stge_oN)XIC(MCP_GY_01_Gripper.Brake_Released)XIO(HMI_Gantry_01_Gripper_PB.2)XIO(HMI_Gantry_01_Gripper_PB.3)MOV(100,MCP_GY_01_Gripper.Application_Mode)XIC(HMI_Gantry_01_Gripper_PB.5)OTE(MCP_GY_01_Gripper.Jog_Pos);
   2: XIC(HMI_Gantry_01_Gripper_PB.1)XIC(MCP_GY_01_Gripper.PwR_Stge_oN)XIC(MCP_GY_01_Gripper.Brake_Released)XIC(HMI_Gantry_01_Gripper_PB.6)MOV(100,MCP_GY_01_Gripper.Application_Mode)OTE(MCP_GY_01_Gripper.Jog_Neg);
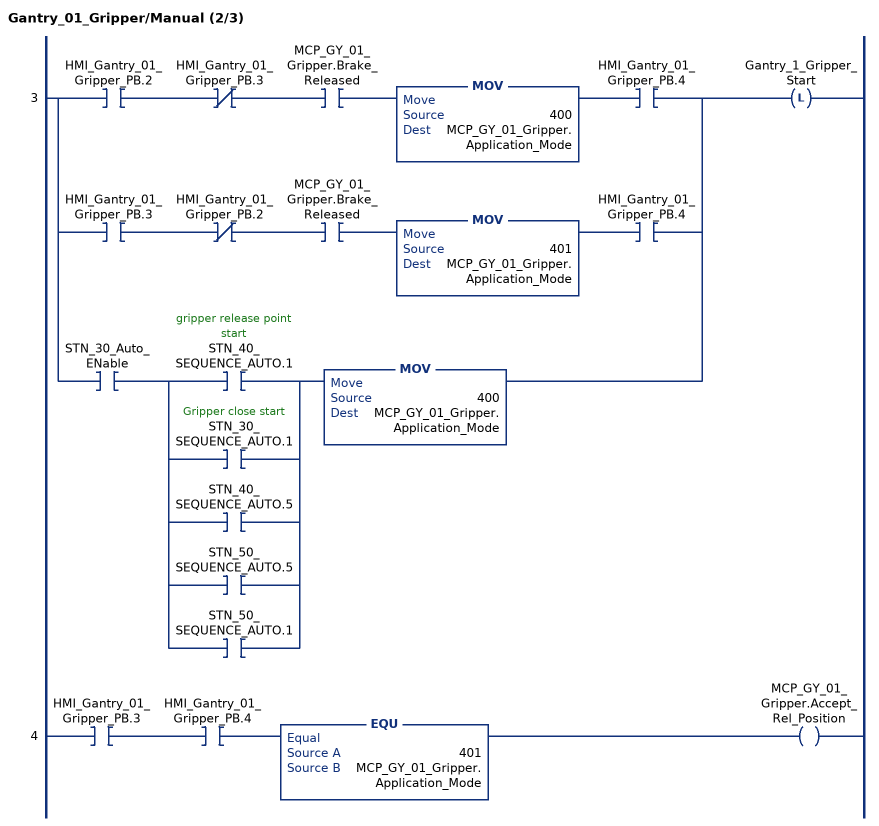
   3: [XIC(HMI_Gantry_01_Gripper_PB.2) XIO(HMI_Gantry_01_Gripper_PB.3) XIC(MCP_GY_01_Gripper.Brake_Released) MOV(400,MCP_GY_01_Gripper.Application_Mode) XIC(HMI_Gantry_01_Gripper_PB.4) ,XIC(HMI_Gantry_01_Gripper_PB.3) XIO(HMI_Gantry_01_Gripper_PB.2) XIC(MCP_GY_01_Gripper.Brake_Released) MOV(401,MCP_GY_01_Gripper.Application_Mode) XIC(HMI_Gantry_01_Gripper_PB.4) ,XIC(STN_30_Auto_ENable) [XIC(STN_40_SEQUENCE_AUTO.1) ,[XIC(STN_30_SEQUENCE_AUTO.1) ,XIC(STN_40_SEQUENCE_AUTO.5) ,XIC(STN_50_SEQUENCE_AUTO.5) ,XIC(STN_50_SEQUENCE_AUTO.1) ] ] MOV(400,MCP_GY_01_Gripper.Application_Mode) ]OTL(Gantry_1_Gripper_Start);
   4: XIC(HMI_Gantry_01_Gripper_PB.3)XIC(HMI_Gantry_01_Gripper_PB.4)EQU(401,MCP_GY_01_Gripper.Application_Mode)OTE(MCP_GY_01_Gripper.Accept_Rel_Position);
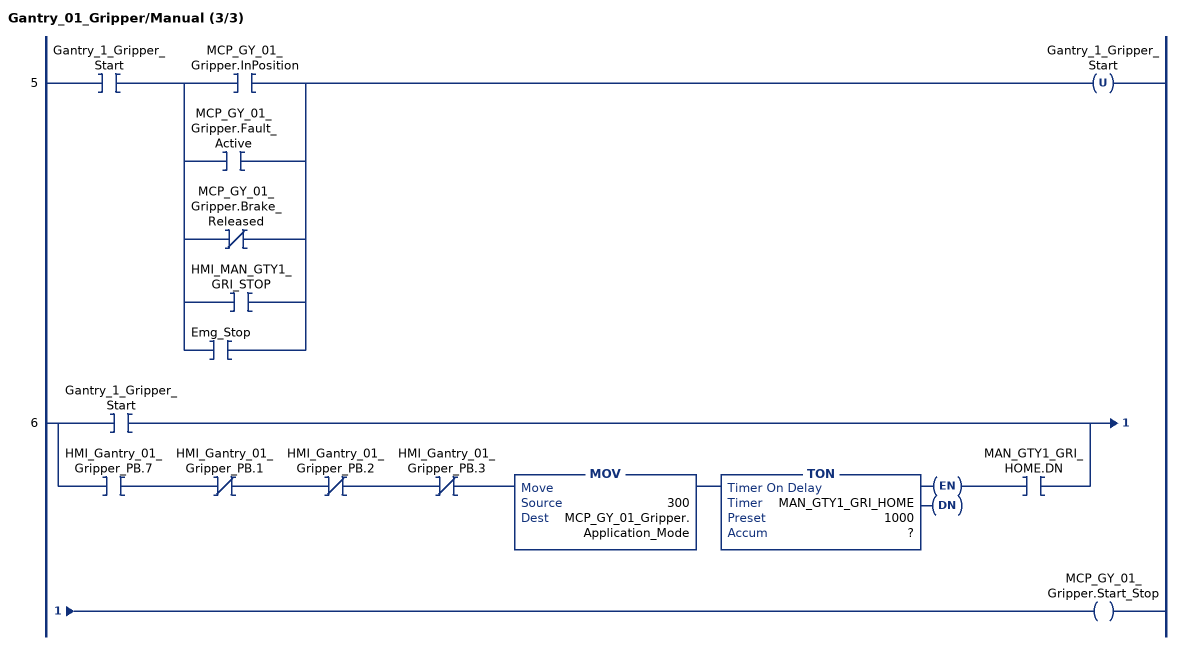
   5: XIC(Gantry_1_Gripper_Start)[XIC(MCP_GY_01_Gripper.InPosition) ,[XIC(MCP_GY_01_Gripper.Fault_Active) ,[XIO(MCP_GY_01_Gripper.Brake_Released) ,[XIC(HMI_MAN_GTY1_GRI_STOP) ,XIC(Emg_Stop) ] ] ] ]OTU(Gantry_1_Gripper_Start);
   6: [XIC(Gantry_1_Gripper_Start) ,XIC(HMI_Gantry_01_Gripper_PB.7) XIO(HMI_Gantry_01_Gripper_PB.1) XIO(HMI_Gantry_01_Gripper_PB.2) XIO(HMI_Gantry_01_Gripper_PB.3) MOV(300,MCP_GY_01_Gripper.Application_Mode) TON(MAN_GTY1_GRI_HOME,?,?) XIC(MAN_GTY1_GRI_HOME.DN) ]OTE(MCP_GY_01_Gripper.Start_Stop);
END_ROUTINE

ROUTINE Servo   (* ladder *)
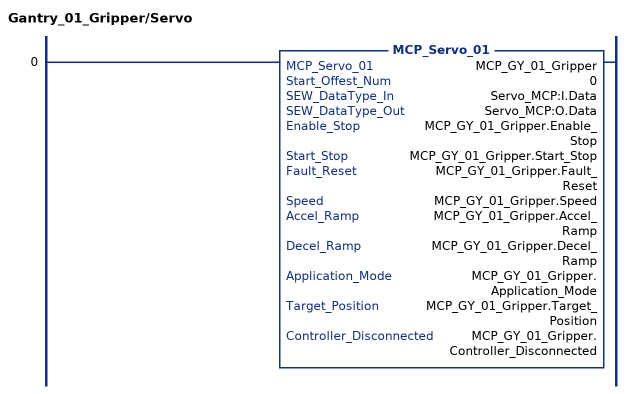
   0: MCP_Servo_01(MCP_GY_01_Gripper,0,Servo_MCP:I.Data,Servo_MCP:O.Data,MCP_GY_01_Gripper.Enable_Stop,MCP_GY_01_Gripper.Start_Stop,MCP_GY_01_Gripper.Fault_Reset,MCP_GY_01_Gripper.Speed,MCP_GY_01_Gripper.Accel_Ramp,MCP_GY_01_Gripper.Decel_Ramp,MCP_GY_01_Gripper.Application_Mode,MCP_GY_01_Gripper.Target_Position,MCP_GY_01_Gripper.Controller_Disconnected);
END_ROUTINE
END_PROGRAM

PROGRAM Gantry_01_Horizontal   (* main routine Main *)

ROUTINE Main   (* ladder *)
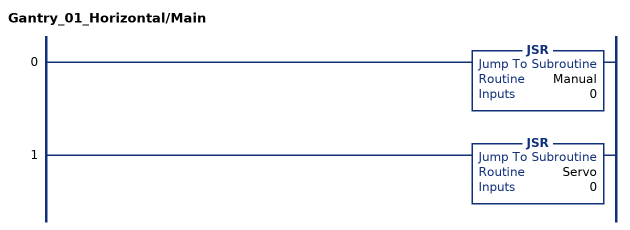
   0: JSR(Manual,0);
   1: JSR(Servo,0);
END_ROUTINE

ROUTINE Manual   (* ladder *)
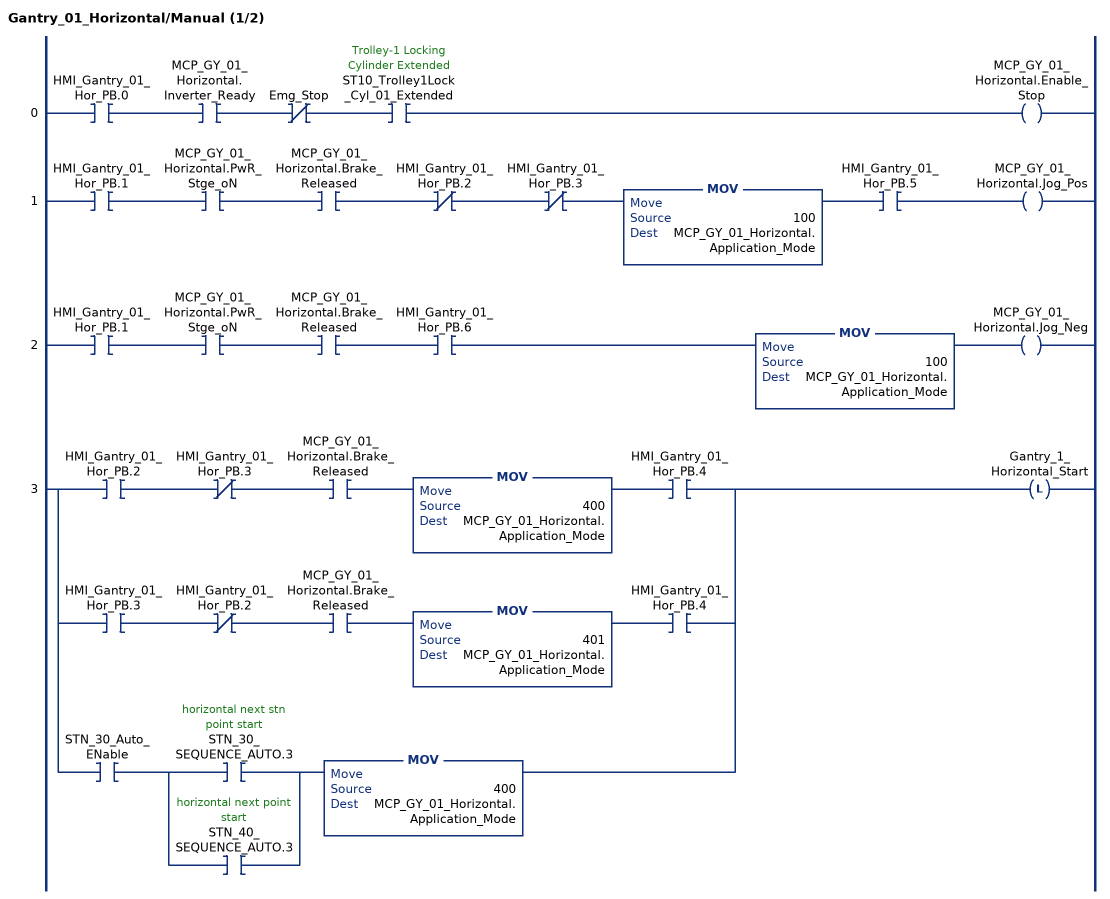
   0: XIC(HMI_Gantry_01_Hor_PB.0)XIC(MCP_GY_01_Horizontal.Inverter_Ready)XIO(Emg_Stop)XIC(ST10_Trolley1Lock_Cyl_01_Extended)OTE(MCP_GY_01_Horizontal.Enable_Stop);
   1: XIC(HMI_Gantry_01_Hor_PB.1)XIC(MCP_GY_01_Horizontal.PwR_Stge_oN)XIC(MCP_GY_01_Horizontal.Brake_Released)XIO(HMI_Gantry_01_Hor_PB.2)XIO(HMI_Gantry_01_Hor_PB.3)MOV(100,MCP_GY_01_Horizontal.Application_Mode)XIC(HMI_Gantry_01_Hor_PB.5)OTE(MCP_GY_01_Horizontal.Jog_Pos);
   2: XIC(HMI_Gantry_01_Hor_PB.1)XIC(MCP_GY_01_Horizontal.PwR_Stge_oN)XIC(MCP_GY_01_Horizontal.Brake_Released)XIC(HMI_Gantry_01_Hor_PB.6)MOV(100,MCP_GY_01_Horizontal.Application_Mode)OTE(MCP_GY_01_Horizontal.Jog_Neg);
   3: [XIC(HMI_Gantry_01_Hor_PB.2) XIO(HMI_Gantry_01_Hor_PB.3) XIC(MCP_GY_01_Horizontal.Brake_Released) MOV(400,MCP_GY_01_Horizontal.Application_Mode) XIC(HMI_Gantry_01_Hor_PB.4) ,[XIC(HMI_Gantry_01_Hor_PB.3) XIO(HMI_Gantry_01_Hor_PB.2) XIC(MCP_GY_01_Horizontal.Brake_Released) MOV(401,MCP_GY_01_Horizontal.Application_Mode) XIC(HMI_Gantry_01_Hor_PB.4) ,XIC(STN_30_Auto_ENable) [XIC(STN_30_SEQUENCE_AUTO.3) ,XIC(STN_40_SEQUENCE_AUTO.3) ] MOV(400,MCP_GY_01_Horizontal.Application_Mode) ] ]OTL(Gantry_1_Horizontal_Start);
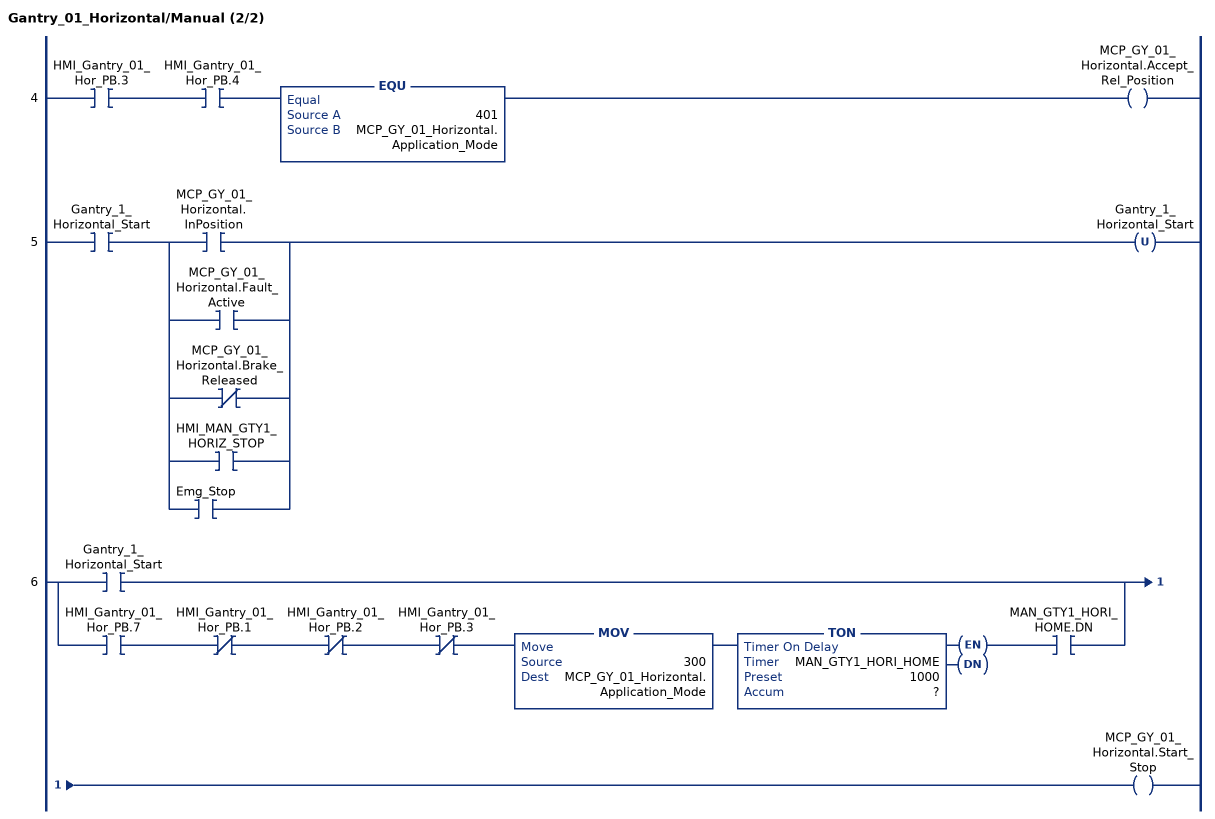
   4: XIC(HMI_Gantry_01_Hor_PB.3)XIC(HMI_Gantry_01_Hor_PB.4)EQU(401,MCP_GY_01_Horizontal.Application_Mode)OTE(MCP_GY_01_Horizontal.Accept_Rel_Position);
   5: XIC(Gantry_1_Horizontal_Start)[XIC(MCP_GY_01_Horizontal.InPosition) ,[XIC(MCP_GY_01_Horizontal.Fault_Active) ,[XIO(MCP_GY_01_Horizontal.Brake_Released) ,[XIC(HMI_MAN_GTY1_HORIZ_STOP) ,XIC(Emg_Stop) ] ] ] ]OTU(Gantry_1_Horizontal_Start);
   6: [XIC(Gantry_1_Horizontal_Start) ,XIC(HMI_Gantry_01_Hor_PB.7) XIO(HMI_Gantry_01_Hor_PB.1) XIO(HMI_Gantry_01_Hor_PB.2) XIO(HMI_Gantry_01_Hor_PB.3) MOV(300,MCP_GY_01_Horizontal.Application_Mode) TON(MAN_GTY1_HORI_HOME,?,?) XIC(MAN_GTY1_HORI_HOME.DN) ]OTE(MCP_GY_01_Horizontal.Start_Stop);
END_ROUTINE

ROUTINE Servo   (* ladder *)
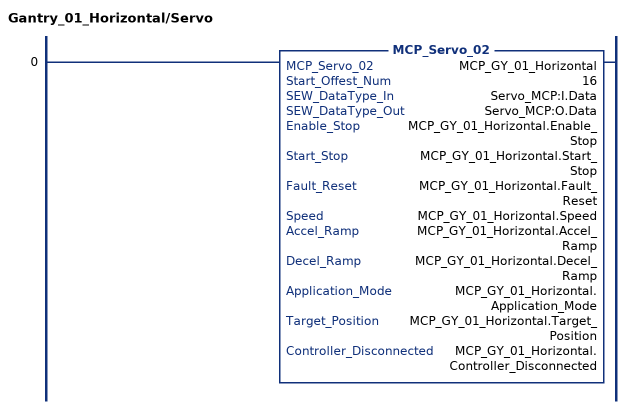
   0: MCP_Servo_02(MCP_GY_01_Horizontal,16,Servo_MCP:I.Data,Servo_MCP:O.Data,MCP_GY_01_Horizontal.Enable_Stop,MCP_GY_01_Horizontal.Start_Stop,MCP_GY_01_Horizontal.Fault_Reset,MCP_GY_01_Horizontal.Speed,MCP_GY_01_Horizontal.Accel_Ramp,MCP_GY_01_Horizontal.Decel_Ramp,MCP_GY_01_Horizontal.Application_Mode,MCP_GY_01_Horizontal.Target_Position,MCP_GY_01_Horizontal.Controller_Disconnected);
END_ROUTINE
END_PROGRAM

PROGRAM Gantry_01_Vertical   (* main routine Main *)

ROUTINE Main   (* ladder *)
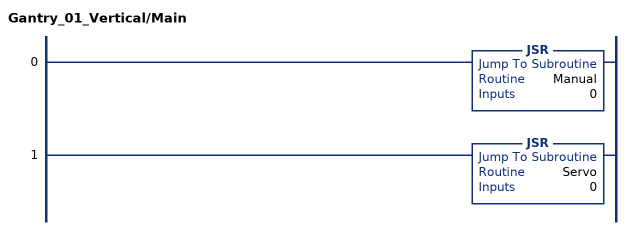
   0: JSR(Manual,0);
   1: JSR(Servo,0);
END_ROUTINE

ROUTINE Manual   (* ladder *)
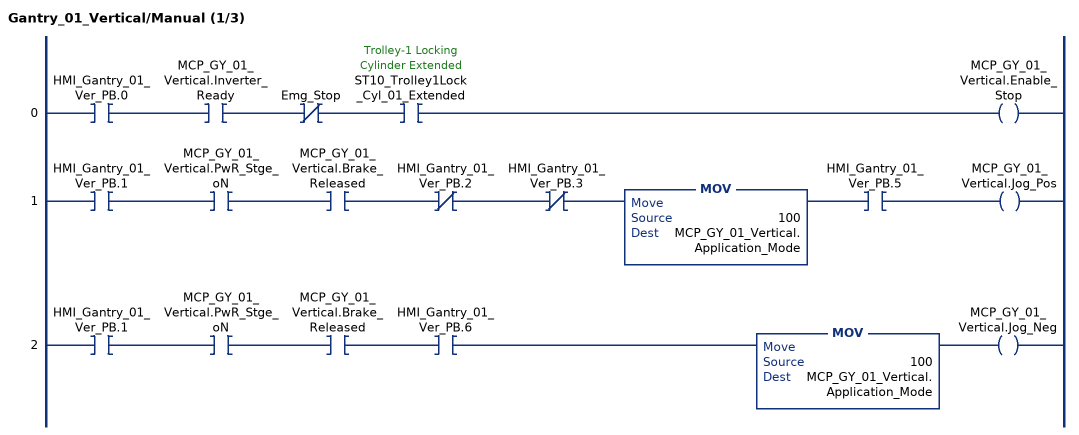
   0: XIC(HMI_Gantry_01_Ver_PB.0)XIC(MCP_GY_01_Vertical.Inverter_Ready)XIO(Emg_Stop)XIC(ST10_Trolley1Lock_Cyl_01_Extended)OTE(MCP_GY_01_Vertical.Enable_Stop);
   1: XIC(HMI_Gantry_01_Ver_PB.1)XIC(MCP_GY_01_Vertical.PwR_Stge_oN)XIC(MCP_GY_01_Vertical.Brake_Released)XIO(HMI_Gantry_01_Ver_PB.2)XIO(HMI_Gantry_01_Ver_PB.3)MOV(100,MCP_GY_01_Vertical.Application_Mode)XIC(HMI_Gantry_01_Ver_PB.5)OTE(MCP_GY_01_Vertical.Jog_Pos);
   2: XIC(HMI_Gantry_01_Ver_PB.1)XIC(MCP_GY_01_Vertical.PwR_Stge_oN)XIC(MCP_GY_01_Vertical.Brake_Released)XIC(HMI_Gantry_01_Ver_PB.6)MOV(100,MCP_GY_01_Vertical.Application_Mode)OTE(MCP_GY_01_Vertical.Jog_Neg);
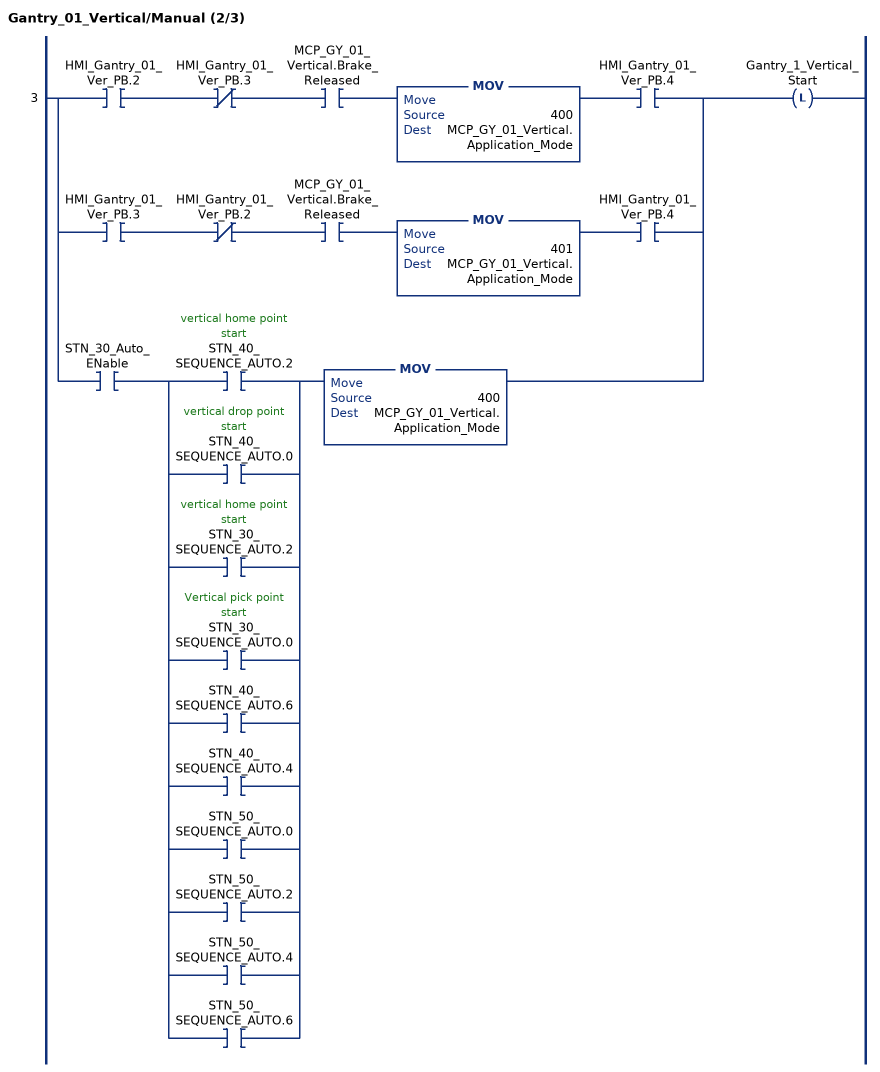
   3: [XIC(HMI_Gantry_01_Ver_PB.2) XIO(HMI_Gantry_01_Ver_PB.3) XIC(MCP_GY_01_Vertical.Brake_Released) MOV(400,MCP_GY_01_Vertical.Application_Mode) XIC(HMI_Gantry_01_Ver_PB.4) ,XIC(HMI_Gantry_01_Ver_PB.3) XIO(HMI_Gantry_01_Ver_PB.2) XIC(MCP_GY_01_Vertical.Brake_Released) MOV(401,MCP_GY_01_Vertical.Application_Mode) XIC(HMI_Gantry_01_Ver_PB.4) ,XIC(STN_30_Auto_ENable) [XIC(STN_40_SEQUENCE_AUTO.2) ,XIC(STN_40_SEQUENCE_AUTO.0) ,XIC(STN_30_SEQUENCE_AUTO.2) ,[XIC(STN_30_SEQUENCE_AUTO.0) ,XIC(STN_40_SEQUENCE_AUTO.6) ,XIC(STN_40_SEQUENCE_AUTO.4) ,XIC(STN_50_SEQUENCE_AUTO.0) ,XIC(STN_50_SEQUENCE_AUTO.2) ,XIC(STN_50_SEQUENCE_AUTO.4) ,XIC(STN_50_SEQUENCE_AUTO.6) ] ] MOV(400,MCP_GY_01_Vertical.Application_Mode) ]OTL(Gantry_1_Vertical_Start);
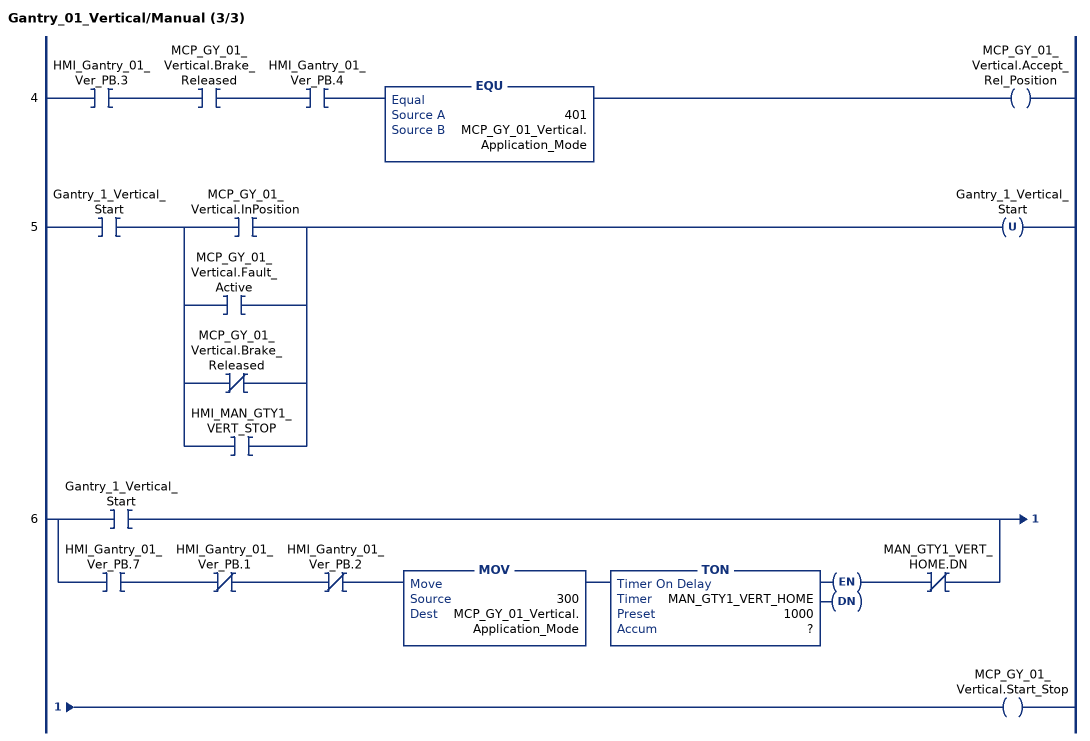
   4: XIC(HMI_Gantry_01_Ver_PB.3)XIC(MCP_GY_01_Vertical.Brake_Released)XIC(HMI_Gantry_01_Ver_PB.4)EQU(401,MCP_GY_01_Vertical.Application_Mode)OTE(MCP_GY_01_Vertical.Accept_Rel_Position);
   5: XIC(Gantry_1_Vertical_Start)[XIC(MCP_GY_01_Vertical.InPosition) ,[XIC(MCP_GY_01_Vertical.Fault_Active) ,[XIO(MCP_GY_01_Vertical.Brake_Released) ,XIC(HMI_MAN_GTY1_VERT_STOP) ] ] ]OTU(Gantry_1_Vertical_Start);
   6: [XIC(Gantry_1_Vertical_Start) ,XIC(HMI_Gantry_01_Ver_PB.7) XIO(HMI_Gantry_01_Ver_PB.1) XIO(HMI_Gantry_01_Ver_PB.2) MOV(300,MCP_GY_01_Vertical.Application_Mode) TON(MAN_GTY1_VERT_HOME,?,?) XIO(MAN_GTY1_VERT_HOME.DN) ]OTE(MCP_GY_01_Vertical.Start_Stop);
END_ROUTINE

ROUTINE Servo   (* ladder *)
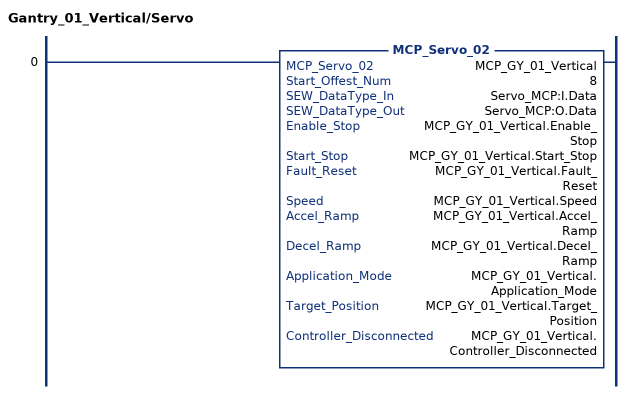
   0: MCP_Servo_02(MCP_GY_01_Vertical,8,Servo_MCP:I.Data,Servo_MCP:O.Data,MCP_GY_01_Vertical.Enable_Stop,MCP_GY_01_Vertical.Start_Stop,MCP_GY_01_Vertical.Fault_Reset,MCP_GY_01_Vertical.Speed,MCP_GY_01_Vertical.Accel_Ramp,MCP_GY_01_Vertical.Decel_Ramp,MCP_GY_01_Vertical.Application_Mode,MCP_GY_01_Vertical.Target_Position,MCP_GY_01_Vertical.Controller_Disconnected);
END_ROUTINE
END_PROGRAM

PROGRAM Gantry_02_Gripper   (* main routine Main *)

ROUTINE Main   (* ladder *)
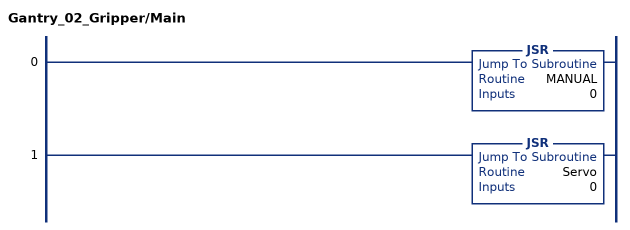
   0: JSR(MANUAL,0);
   1: JSR(Servo,0);
END_ROUTINE

ROUTINE MANUAL   (* ladder *)
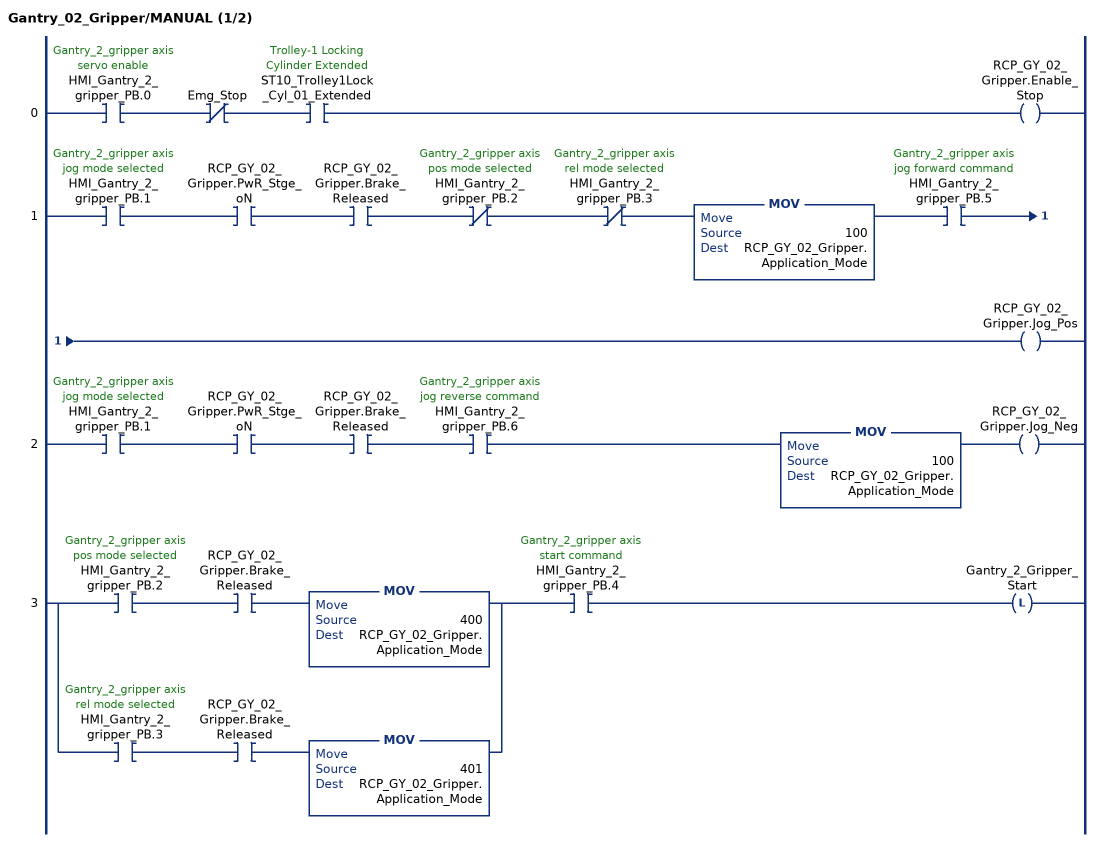
   0: XIC(HMI_Gantry_2_gripper_PB.0)XIO(Emg_Stop)XIC(ST10_Trolley1Lock_Cyl_01_Extended)OTE(RCP_GY_02_Gripper.Enable_Stop);
   1: XIC(HMI_Gantry_2_gripper_PB.1)XIC(RCP_GY_02_Gripper.PwR_Stge_oN)XIC(RCP_GY_02_Gripper.Brake_Released)XIO(HMI_Gantry_2_gripper_PB.2)XIO(HMI_Gantry_2_gripper_PB.3)MOV(100,RCP_GY_02_Gripper.Application_Mode)XIC(HMI_Gantry_2_gripper_PB.5)OTE(RCP_GY_02_Gripper.Jog_Pos);
   2: XIC(HMI_Gantry_2_gripper_PB.1)XIC(RCP_GY_02_Gripper.PwR_Stge_oN)XIC(RCP_GY_02_Gripper.Brake_Released)XIC(HMI_Gantry_2_gripper_PB.6)MOV(100,RCP_GY_02_Gripper.Application_Mode)OTE(RCP_GY_02_Gripper.Jog_Neg);
   3: [XIC(HMI_Gantry_2_gripper_PB.2) XIC(RCP_GY_02_Gripper.Brake_Released) MOV(400,RCP_GY_02_Gripper.Application_Mode) ,XIC(HMI_Gantry_2_gripper_PB.3) XIC(RCP_GY_02_Gripper.Brake_Released) MOV(401,RCP_GY_02_Gripper.Application_Mode) ]XIC(HMI_Gantry_2_gripper_PB.4)OTL(Gantry_2_Gripper_Start);
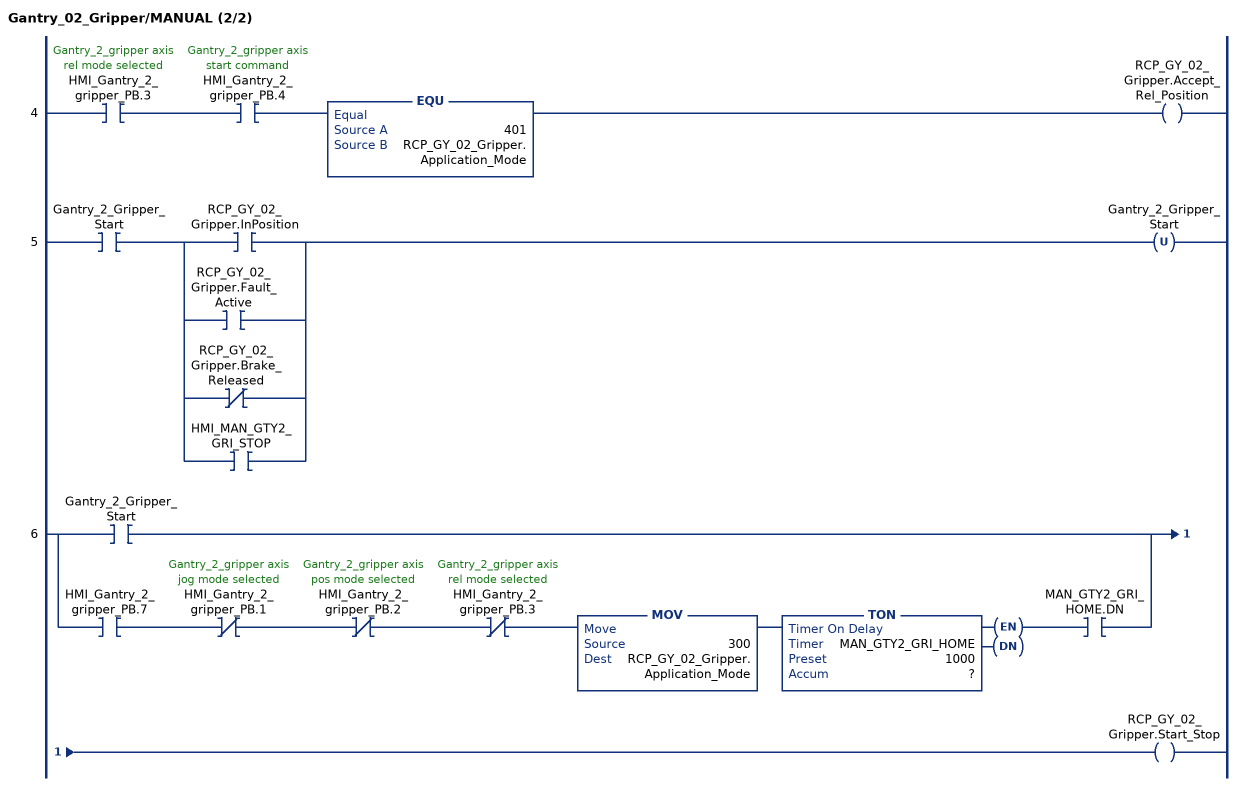
   4: XIC(HMI_Gantry_2_gripper_PB.3)XIC(HMI_Gantry_2_gripper_PB.4)EQU(401,RCP_GY_02_Gripper.Application_Mode)OTE(RCP_GY_02_Gripper.Accept_Rel_Position);
   5: XIC(Gantry_2_Gripper_Start)[XIC(RCP_GY_02_Gripper.InPosition) ,[XIC(RCP_GY_02_Gripper.Fault_Active) ,[XIO(RCP_GY_02_Gripper.Brake_Released) ,XIC(HMI_MAN_GTY2_GRI_STOP) ] ] ]OTU(Gantry_2_Gripper_Start);
   6: [XIC(Gantry_2_Gripper_Start) ,XIC(HMI_Gantry_2_gripper_PB.7) XIO(HMI_Gantry_2_gripper_PB.1) XIO(HMI_Gantry_2_gripper_PB.2) XIO(HMI_Gantry_2_gripper_PB.3) MOV(300,RCP_GY_02_Gripper.Application_Mode) TON(MAN_GTY2_GRI_HOME,?,?) XIC(MAN_GTY2_GRI_HOME.DN) ]OTE(RCP_GY_02_Gripper.Start_Stop);
END_ROUTINE

ROUTINE Servo   (* ladder *)
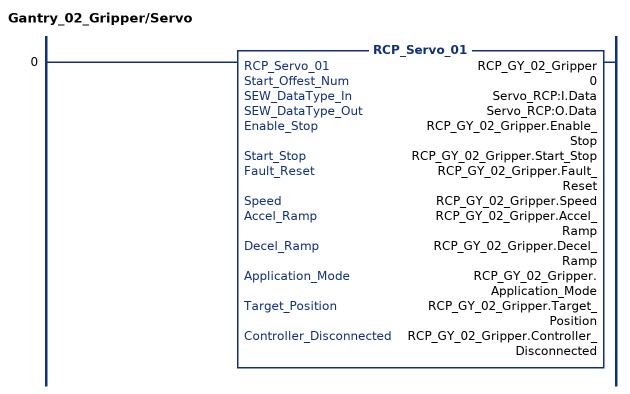
   0: RCP_Servo_01(RCP_GY_02_Gripper,0,Servo_RCP:I.Data,Servo_RCP:O.Data,RCP_GY_02_Gripper.Enable_Stop,RCP_GY_02_Gripper.Start_Stop,RCP_GY_02_Gripper.Fault_Reset,RCP_GY_02_Gripper.Speed,RCP_GY_02_Gripper.Accel_Ramp,RCP_GY_02_Gripper.Decel_Ramp,RCP_GY_02_Gripper.Application_Mode,RCP_GY_02_Gripper.Target_Position,RCP_GY_02_Gripper.Controller_Disconnected);
END_ROUTINE
END_PROGRAM
